// TIA Portal project "Tank Doldurup Boşaltma" (V15)
// Vorlageprojekt für das Buch mit Zielsystem S7-1200

(* hardware
DEVICE "S7-1200-Station_1"  S7-1200 Station
   slot 0: "Baugruppenträger_0"  Rack  V1.0
   slot 1: "PLC_1"  CPU 1211C DC/DC/DC  6ES7 211-1AE40-0XB0  V4.1
*)

// ===== PLC "PLC_1"  CPU 1211C DC/DC/DC =====

VAR_GLOBAL   // PLC tag table "Standard-Variablentabelle"
   "Fill" AT %I0.0 : Bool;
   "Yardımcı_Röle" AT %M0.0 : Bool;
   "Fill_Valve" AT %Q0.0 : Bool;
   "Fill_Value" AT %Q0.1 : Bool;
   "Discharge" AT %I0.1 : Bool;
   "Yardımcı_Röle_2" AT %M0.1 : Bool;
   "Discharge_Valve" AT %Q0.2 : Bool;
   "Discharge_Value" AT %Q0.3 : Bool;
   "Tag_1" AT %QD30 : Time;
   "Tag_2" AT %QD34 : Time;
END_VAR

// folder: System blocks/Program resources

DATA_BLOCK "Timer_1"   // DB1
{ S7_Optimized_Access := 'TRUE' }
AUTHOR : Simatic
FAMILY : IEC
NAME : IEC_TMR
VERSION : 1.0
// stored: InstanceOfName IEC_TIMER
"IEC_TIMER"
BEGIN
END_DATA_BLOCK

DATA_BLOCK "Timer_2"   // DB2
{ S7_Optimized_Access := 'TRUE' }
AUTHOR : Simatic
FAMILY : IEC
NAME : IEC_TMR
VERSION : 1.0
// stored: InstanceOfName IEC_TIMER
"IEC_TIMER"
BEGIN
END_DATA_BLOCK

// folder: (top level)

FUNCTION "MHJ-PLC-Lab-Function-S71200" : Void   // FC9000, SCL
{ S7_Optimized_Access := 'TRUE' }
VERSION : 0.1
   VAR_TEMP
      rdTimeReturn : Int;
      outputTime : DTL;
      SyncVal : Byte;
      forVal : Int;
      forVal_2 : Int;
      Value : Byte;
   END_VAR
   VAR CONSTANT
      CompVal : Byte := 16#34;
      Value_01 : Byte := 16#11;
      Value_01_DW : DWord := 16#A165_D992;
      Value_02_DW : DWord := 16#58BE_4401;
   END_VAR
BEGIN

   #Value:=PEEK(area := 16#82,
        dbNumber := 0,
        byteOffset := 511);
   #Value := #Value + 1;

   POKE(area := 16#82,
        dbNumber := 0,
        byteOffset := 511,
        value := #Value);

   POKE(area:=16#81,
        dbNumber:=0,
        byteOffset:=1016,
        value:=#Value_01_DW);
   POKE(area := 16#81,
        dbNumber := 0,
        byteOffset := 1020,
        value := #Value_02_DW);

   POKE(area := 16#81,
        dbNumber := 0,
        byteOffset := 511,
        value := B#16#00);

   FOR #forVal := 0 TO 120 DO
       FOR #forVal_2:=0 TO 10 DO
           #rdTimeReturn:=RD_SYS_T(#outputTime);
           #rdTimeReturn := WR_SYS_T(#outputTime);
           #rdTimeReturn := RD_SYS_T(#outputTime);
           #rdTimeReturn := WR_SYS_T(#outputTime);
       END_FOR;
       #SyncVal:= PEEK(area := 16#81,
                      dbNumber := 0,
                      byteOffset := 511);
       IF #SyncVal = #CompVal THEN
          GOTO M_1;
       END_IF;
   END_FOR;
   RETURN;

   M_1:
   POKE(area := 16#81,
        dbNumber := 0,
        byteOffset := 511,
        value := B#16#0);
END_FUNCTION

ORGANIZATION_BLOCK "Main"   // OB1, LAD, ProgramCycle
TITLE = "Main Program Sweep (Cycle)"
{ S7_Optimized_Access := 'TRUE' }
VERSION : 0.1
   VAR_INPUT
      Initial_Call : Bool;   // Initial call of this OB
      Remanence : Bool;   // =True, if remanent data are available
   END_VAR
BEGIN

REGION Network 1: Konnektierungsbaustein für PLC-Lab
   // Im Netzwerk 1 wird der Konnektierungsbaustein für PLC-Lab aufgerufen.
   // Dieser Aufruf darf nicht entfernt werden!
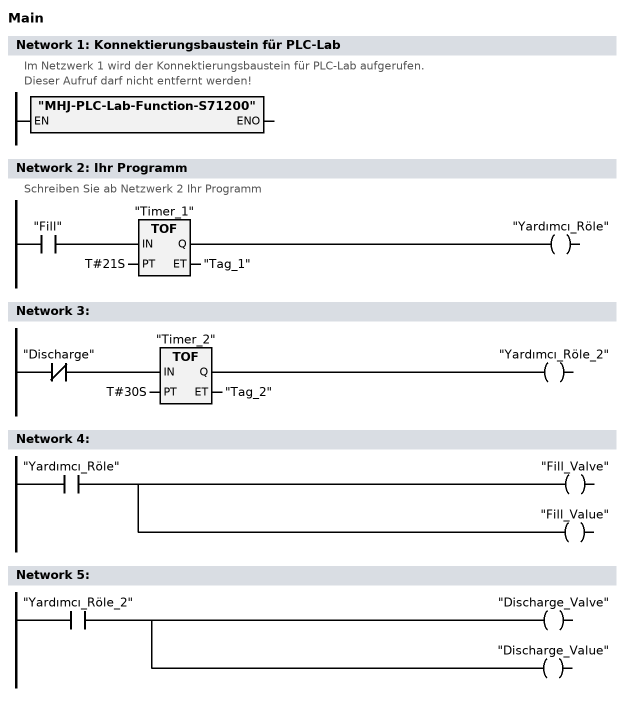
   RUNG wire#powerrail
      "MHJ-PLC-Lab-Function-S71200"()
   END_RUNG
   // the same network as SCL:
   "MHJ-PLC-Lab-Function-S71200"();
END_REGION

REGION Network 2: Ihr Programm
   // Schreiben Sie ab Netzwerk 2 Ihr Programm
   "Timer_1".TOF(IN := "Fill", PT := T#21S, ET => "Tag_1");
   "Yardımcı_Röle" := "Timer_1".Q;
END_REGION

REGION Network 3
   "Timer_2".TOF(IN := NOT "Discharge", PT := T#30S, ET => "Tag_2");
   "Yardımcı_Röle_2" := "Timer_2".Q;
END_REGION

REGION Network 4
   RUNG wire#powerrail
      Contact( "Yardımcı_Röle" )
      wire#w1
      Coil( "Fill_Valve" )
   END_RUNG
   RUNG wire#w1
      Coil( "Fill_Value" )
   END_RUNG
   // the same network as SCL:
   "Fill_Valve" := "Yardımcı_Röle";
   "Fill_Value" := "Yardımcı_Röle";
END_REGION

REGION Network 5
   RUNG wire#powerrail
      Contact( "Yardımcı_Röle_2" )
      wire#w1
      Coil( "Discharge_Valve" )
   END_RUNG
   RUNG wire#w1
      Coil( "Discharge_Value" )
   END_RUNG
   // the same network as SCL:
   "Discharge_Valve" := "Yardımcı_Röle_2";
   "Discharge_Value" := "Yardımcı_Röle_2";
END_REGION
END_ORGANIZATION_BLOCK